// TIA Portal V19 export
DATA_BLOCK "DB_Arduino_Tcp_Connect"   // DB10
{ S7_Optimized_Access := 'TRUE' }
// stored: MemoryReserve 100
   VAR
      MB_Arduino_Write : TCON_IP_v4;
      MB_Arduino_Read : TCON_IP_v4;
      MB_Arduino_Disconnect { S7_SetPoint := 'True'} : Bool;
      MB_Arduino_Req : Bool;
      MB_Arduino_Error : Bool;
      MB_Arduino_Done : Bool;
      MB_Arduino_Busy : Bool;
      MB_Arduino_Status : Word;
      MB_Arduino_Write_Busy : Bool;
      MB_Arduino_Write_Done : Bool;
      MB_Arduino_Write_Error : Bool;
      MB_Arduino_Write_Req : Bool;
      MB_Arduino_Write_Disconnect : Bool;
      MB_Arduino_Write_Status : Word;
   END_VAR
BEGIN
   MB_Arduino_Write.InterfaceId := 64;
   MB_Arduino_Write.ID := 16#1;
   MB_Arduino_Write.ConnectionType := 16#0B;
   MB_Arduino_Write.ActiveEstablished := 1;
   MB_Arduino_Write.RemoteAddress.ADDR[1] := 16#C0;
   MB_Arduino_Write.RemoteAddress.ADDR[2] := 16#A8;
   MB_Arduino_Write.RemoteAddress.ADDR[3] := 16#1;
   MB_Arduino_Write.RemoteAddress.ADDR[4] := 16#3D;
   MB_Arduino_Write.RemotePort := 502;
   MB_Arduino_Read.InterfaceId := 64;
   MB_Arduino_Read.ID := 16#1;
   MB_Arduino_Read.ConnectionType := 16#0B;
   MB_Arduino_Read.ActiveEstablished := 1;
   MB_Arduino_Read.RemoteAddress.ADDR[1] := 16#C0;
   MB_Arduino_Read.RemoteAddress.ADDR[2] := 16#A8;
   MB_Arduino_Read.RemoteAddress.ADDR[3] := 16#1;
   MB_Arduino_Read.RemoteAddress.ADDR[4] := 16#3D;
   MB_Arduino_Read.RemotePort := 502;
END_DATA_BLOCK
